Staubli VAL3: tskCollision.pgx

program tskCollision()
  local num LnDistance
  local point LpHere
  local point LpPark
  local bool l_bPPSint
  local bool l_bStageint
  local num l_nLastChange
  local num l_nOldHeartbeat
  local num l_nTime
  local string sReturn
begin
  //header begin
  // PROGRAM tskColision()

  //header end


  do

    if dioGet(dCollisionSens)>0
      nColision=1
    else
      nColision=0
    endIf

    // logMsg(toString("",nColision))

    if dioGet(dCollisionSens)==0

      stopMove()
      resetMotion()
      disablePower()

      popUpMsg("COLLISION DETECTED!")

    endIf



  until false




end
